// TwinCAT 3 PLC project PLC_WeldingRobot
// ProgramVersion: 3.1.4026.26
// libraries:
//   Tc2_Standard, * (Beckhoff Automation GmbH)
//   Tc2_System, * (Beckhoff Automation GmbH)
// project tree:
//   DUTs/ E_AutomaticMode.TcDUT, E_ManualMode.TcDUT, E_Mode.TcDUT, E_SemiAutomatic.TcDUT, ST_Order.TcDUT
//   / PlcTask.TcTTO
//   POUs/ FB_Robot.TcPOU (not stored), FB_Stepper.TcPOU (not stored), MAIN.TcPOU
// real-time tasks:
//   TASK PlcTask: cycle T#10ms, priority 20, ADS port 350
// I/O:
//   DEVICE Device 1 (EtherCAT), AmsNetId 192.168.2.107.2.1
//     Term 1 (EK1200) [EK1200-5000 EtherCAT Power supply (2A E-Bus)]
//       Term 2 (EL1004) [EL1004 4Ch. Dig. Input 24V, 3ms]
//       Term 3 (EL3204) [EL3204 4Ch. Ana. Input PT100 (RTD)]
//       Term 4 (EL9508) [EL9508 Power supply terminal 8V]
//       Term 5 (EL2624) [EL2624 4Ch. Relay Output, NO (125V AC / 30V DC)]
//       Term 6 (EL2612) [EL2612 2Ch. Relay Output, CO (125V AC / 30V DC)]
//       Term 7 (EL9011) [EL9011 End Terminal]
// variable links:
//   PLC_WeldingRobot/PLC_WeldingRobot Instance <-> Device 1 (EtherCAT)/Term 1 (EK1200)/Term 2 (EL1004)
//     PlcTask Inputs/MAIN.fbRobot.fbStepper.bHomingSensor <-> Channel 1/Input
//     PlcTask Inputs/MAIN.fbRobot.fbStepper.bStepSensor <-> Channel 2/Input
//   PLC_WeldingRobot/PLC_WeldingRobot Instance <-> Device 1 (EtherCAT)/Term 1 (EK1200)/Term 5 (EL2624)
//     PlcTask Outputs/MAIN.fbRobot.bWeld <-> Channel 1/Output
//   PLC_WeldingRobot/PLC_WeldingRobot Instance <-> Device 1 (EtherCAT)/Term 1 (EK1200)/Term 6 (EL2612)
//     PlcTask Outputs/MAIN.fbRobot.fbStepper.bMoveBw <-> Channel 2/Output
//     PlcTask Outputs/MAIN.fbRobot.fbStepper.bMoveFw <-> Channel 1/Output

CONFIGURATION PLC_WeldingRobot
    RESOURCE PLC ON TwinCAT3
        TASK PlcTask(INTERVAL := T#10ms, PRIORITY := 20);
        PROGRAM MAIN WITH PlcTask : MAIN;
    END_RESOURCE
END_CONFIGURATION

// ---- DUTs/E_AutomaticMode.TcDUT
TYPE E_AutomaticMode :
(
	eAuto_reset,
	eAuto_ready,
	eAuto_searchOrder,
	eAuto_noOrder,
	eAuto_approachPosition,
	eAuto_weld
);
END_TYPE

// ---- DUTs/E_ManualMode.TcDUT
TYPE E_ManualMode :
(
	eManual_nothing := 0,
	eManual_backward,
	eManual_forward,
	eManual_weld,
	eManual_error
);
END_TYPE

// ---- DUTs/E_Mode.TcDUT
TYPE E_Mode :
(
	eMode_Initial,
	eMode_Secure,
	eMode_Reset,
	eMode_Stop,
	eMode_Manual,
	eMode_SemiAutomatic,
	eMode_FullyAutomatic
);
END_TYPE

// ---- DUTs/E_SemiAutomatic.TcDUT
TYPE E_SemiAutomatic :
(
	eSemi_ready := 0,
	eSemi_wayThere,
	eSemi_weld,
	eSemi_wayBack
);
END_TYPE

// ---- DUTs/ST_Order.TcDUT
TYPE ST_Order :
STRUCT
	nTargetTable	: INT;
	tWeldingTime	: TIME := T#2S;
	bDone			: BOOL;
	bIsValid		: BOOL;
	bWeld			: BOOL := TRUE;
END_STRUCT
END_TYPE

// ---- POUs/MAIN.TcPOU
PROGRAM MAIN
VAR
	fbRobot		: FB_Robot;
END_VAR

fbRobot.Cycle();

END_PROGRAM
